{attribute addProperty BoxType "EL1918-0000-0016"}
{attribute addProperty Id "FSOEAT %I*FSOE_046154CD567"}
{attribute addProperty CRC "1261566923"}
{attribute addProperty SizeInBites "56"}
{attribute addProperty SizeInBytes "7"}
TYPE FSoE_Inputs_4B31FBCB :
STRUCT
	{attribute addProperty Name "FSOE"}
	FSOE AT %I* : FSOE_046154CD;
END_STRUCT
END_TYPE

(* stored: Version 1.2.0.0, ProductVersion 3.1.4024.9
   DUT FSoE_Inputs_4B31FBCB: Id {22bf6cb2-7414-46e8-bc69-0bb795a7a8f7} *)
